(*
    In this testsuite we are running the same testcase over two cycles, and thus calling every assert method twice.
    This is in order to verify that we don't print every FAILED assert twice.
*)
FUNCTION_BLOCK FB_AssertEveryFailedTestTwice EXTENDS TcUnit.FB_TestSuite
VAR
    AssertCount : USINT := 0;
END_VAR

TwiceAssertCall();

METHOD PRIVATE TwiceAssertCall
VAR
    aANY : INT := 55;
    bANY : INT := 77;

    aBOOL : BOOL := TRUE;
    bBOOL : BOOL := FALSE;

    aBYTE : BYTE := 16#AB;
    bBYTE : BYTE := 16#BA;

    aDATE : DATE := DATE#1996-05-06;
    bDATE : DATE := DATE#2019-01-20;

    aDATE_AND_TIME : DATE_AND_TIME := DATE_AND_TIME#1996-05-06-15:36:30;
    bDATE_AND_TIME : DATE_AND_TIME := DATE_AND_TIME#1972-03-29-00:00:00;

    aDINT : DINT := 4444;
    bDINT : DINT := 3333;

    aDWORD : DWORD := 16#AAAAAAAA;
    bDWORD : DWORD := 16#BBBBBBBB;

    aINT : INT := 30000;
    bINT : INT := 32000;

    aLINT : LINT := 50000;
    bLINT : LINT := 50001;

    aLREAL : LREAL := 33.3;
    bLREAL : LREAL := 44.4;

    aLTIME : LTIME := LTIME#213503D23H34M33S709MS551US615NS;
    bLTIME : LTIME := LTIME#1000D15H23M12S34MS2US44NS;

    aLWORD : LWORD := 16#AAAAAAAAAAAAAAAA;
    bLWORD : LWORD := 16#BBBBBBBBBBBBBBBB;

    aREAL : REAL := 44.4;
    bREAL : REAL := 22.2;

    aSINT : SINT := 99;
    bSINT : SINT := 10;

    aSTRING : STRING := 'Hello world';
    bSTRING : STRING := 'Hey there';

    aUDINT : UDINT := 249494994;
    bUDINT : UDINT := 1223;

    aUINT : UINT := 3444;
    bUINT : UINT := 3445;

    aULINT : ULINT := 789234475;
    bULINT : ULINT := 34523327234;

    aUSINT : USINT := 34;
    bUSINT : USINT := 36;

    aTIME : TIME := T#12H34M15S10MS;
    bTIME : TIME := T#11H34M13S244MS;

    aTIME_OF_DAY : TIME_OF_DAY := TIME_OF_DAY#15:36:30.123;
    bTIME_OF_DAY : TIME_OF_DAY := TIME_OF_DAY#06:21:11.492;

    aWORD : WORD := 16#ABCD;
    bWORD : WORD := 16#89EF;

	aWSTRING : WSTRING := "åäöĦ";
    bWSTRING : WSTRING := "åäöŅ";
END_VAR
TEST('TwiceAssertCall');

AssertEquals(Expected := aANY,
             Actual := bANY,
             Message := 'Not equal ANY');

AssertEquals_BOOL(Expected := aBOOL,
                  Actual := bBOOL,
                  Message := 'Not equal BOOL');

AssertEquals_BYTE(Expected := aBYTE,
                  Actual := bBYTE,
                  Message := 'Not equal BYTE');

AssertEquals_DATE(Expected := aDATE,
                  Actual := bDATE,
                  Message := 'Not equal DATE');

AssertEquals_DATE_AND_TIME(Expected := aDATE_AND_TIME,
                           Actual := bDATE_AND_TIME,
                           Message := 'Not equal DATE_AND_TIME');

AssertEquals_DINT(Expected := aDINT,
                  Actual := bDINT,
                  Message := 'Not equal DINT');

AssertEquals_DWORD(Expected := aDWORD,
                   Actual := bDWORD,
                   Message := 'Not equal DWORD');

AssertEquals_INT(Expected := aINT,
                 Actual := bINT,
                 Message := 'Not equal INT');

AssertEquals_LINT(Expected := aLINT,
                  Actual := bLINT,
                  Message := 'Not equal LINT');

AssertEquals_LREAL(Expected := aLREAL,
                   Actual := bLREAL,
                   Delta := 0.1,
                   Message := 'Not equal LREAL');

AssertEquals_LTIME(Expected := aLTIME,
                   Actual := bLTIME,
                   Message := 'Not equal LTIME');

AssertEquals_LWORD(Expected := aLWORD,
                   Actual := bLWORD,
                   Message := 'Not equal LWORD');

AssertEquals_REAL(Expected := aREAL,
                  Actual := bREAL,
                  Delta := 0.1,
                  Message := 'Not equal REAL');

AssertEquals_SINT(Expected := aSINT,
                  Actual := bSINT,
                  Message := 'Not equal SINT');

AssertEquals_STRING(Expected := aSTRING,
                    Actual := bSTRING,
                    Message := 'Not equal STRING');

AssertEquals_UDINT(Expected := aUDINT,
                   Actual := bUDINT,
                   Message := 'Not equal UDINT');

AssertEquals_UINT(Expected := aUINT,
                  Actual := bUINT,
                  Message := 'Not equal UINT');

AssertEquals_ULINT(Expected := aULINT,
                   Actual := bULINT,
                   Message := 'Not equal ULINT');

AssertEquals_USINT(Expected := aUSINT,
                   Actual := bUSINT,
                   Message := 'Not equal USINT');

AssertEquals_TIME(Expected := aTIME,
                  Actual := bTIME,
                  Message := 'Not equal TIME');

AssertEquals_TIME_OF_DAY(Expected := aTIME_OF_DAY,
                         Actual := bTIME_OF_DAY,
                         Message := 'Not equal TIME_OF_DAY');

AssertEquals_WORD(Expected := aWORD,
                  Actual := bWORD,
                  Message := 'Not equal WORD');

AssertEquals_WSTRING(Expected := aWSTRING,
                     Actual := bWSTRING,
                     Message := 'Not equal WSTRING');

AssertCount := AssertCount + 1;
IF AssertCount = 2 THEN
    TEST_FINISHED();
END_IF
END_METHOD

END_FUNCTION_BLOCK

(* stored: Version 1.1.0.1
   POU FB_AssertEveryFailedTestTwice: Id {3bea6e4d-8d08-467b-90da-24a784807eae}, SpecialFunc None
   Method TwiceAssertCall: Id {69d3987a-7ce5-4206-ac7a-879b67c9a54d} *)
